{attribute addProperty BoxType "EL2014-0000-0016"}
{attribute addProperty Id "OutputBIT10.1251"}
{attribute addProperty CRC "3556683513"}
{attribute addProperty SizeInBites "1"}
{attribute addProperty SizeInBytes "0.125"}
{warning 'Size of this structure is not a multiple of 8 bits!!!'}
TYPE Channel_D3FEAEF9 :
STRUCT
	{attribute addProperty Name "Output"}
	Output : BIT;
END_STRUCT
END_TYPE

(* stored: Version 1.2.0.0, ProductVersion 3.1.4024.9
   DUT Channel_D3FEAEF9: Id {b7ed7b50-e153-4e7e-b4a5-ec7ac1bbd389} *)
